FUNCTION_BLOCK ABSTRACT TcoEcatComponent EXTENDS TcoCore.TcoComponent IMPLEMENTS ITcoEcatComponent
VAR_INPUT
    AdsAddr : AMSADDR;
END_VAR
VAR_OUTPUT
END_VAR
VAR
    //*	{attribute addProperty Name "<#Ecat slave state#>"}
    _ecatState : TcoEcatSlaveState(THIS^);
    {attribute 'hide'}
    _sb : TcoCore.StringBuilder;
END_VAR

_ecatState(AdsAddr := AdsAddr);

PROPERTY PUBLIC EcatState : REFERENCE TO TcoEcatSlaveState
GET
EcatState REF= _ecatState;
END_GET
END_PROPERTY

METHOD Restore : ITcoRestorable
VAR_INPUT
END_VAR
_ecatState.Restore();
END_METHOD

METHOD PROTECTED ServiceMode
VAR_INPUT
END_VAR
END_METHOD

END_FUNCTION_BLOCK

(* stored: Version 1.1.0.1, ProductVersion 3.1.4024.11
   POU TcoEcatComponent: Id {14578b19-d1f3-05a5-0327-551bd0348995}, SpecialFunc None
   Folder Public: Id {38e602a5-760f-0e19-1e22-c3acdaaaa854}
   Property EcatState: Id {0a3da69a-83fa-0ae4-0ad4-970396b43f33}
   Get Get: Id {592fa616-451a-073c-2edb-ebfaa10abd18}
   Method Restore: Id {53c9e61d-5af5-072a-2b96-47f256b25f6f}
   Method ServiceMode: Id {7e892b4f-04c3-0d7b-0ebf-779003e20c83} *)
